// SIMATIC S7-200 SMART project (STEP 7-Micro/WIN SMART), CPU ST40

SYMBOL_TABLE Table 1
Counter_1        C1
CON_Done         M0.0
CON_Busy         M0.1
CON_Error        M0.2
CON_Stat         MB1
SEND_Done        M2.0
SEND_Busy        M2.1
SEND_Error       M2.2
SEND_Stat        MB3
END_SYMBOL_TABLE

SYMBOL_TABLE System Symbols
Always_On        SM0.0    // Always ON
First_Scan_On    SM0.1    // ON for the first scan cycle only
Clock_1s         SM0.5    // Clock pulse that is ON for 0.5 s, OFF for 0.5 s, for a duty cycle time of 1 s.
END_SYMBOL_TABLE

ORGANIZATION_BLOCK MAIN:OB1
TITLE=Program Comments
BEGIN
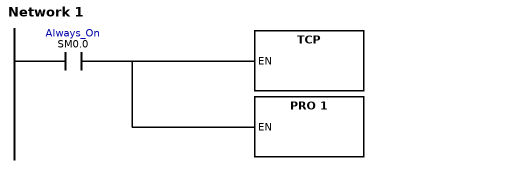
Network 1
LD     Always_On:SM0.0
CALL   TCP:SBR12
CALL   PRO 1:SBR0
END_ORGANIZATION_BLOCK

SUBROUTINE_BLOCK PRO 1:SBR0
TITLE=Subroutine Comments
BEGIN
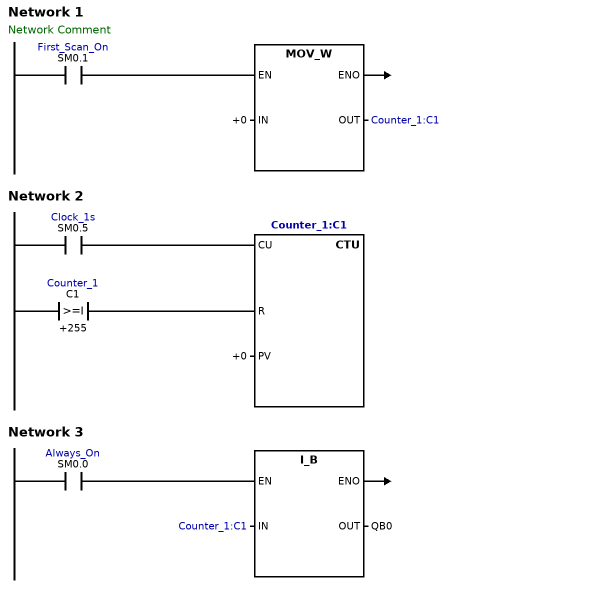
Network 1
// Network Comment
LD     First_Scan_On:SM0.1
MOVW   +0, Counter_1:C1
Network 2
LD     Clock_1s:SM0.5
LDW>=  Counter_1:C1, +255
CTU    Counter_1:C1, +0
Network 3
LD     Always_On:SM0.0
ITB    Counter_1:C1, QB0
END_SUBROUTINE_BLOCK

// SBR10: protected block, not included

// SBR11: protected block, not included

SUBROUTINE_BLOCK TCP:SBR12
TITLE=Subroutine Comments
BEGIN
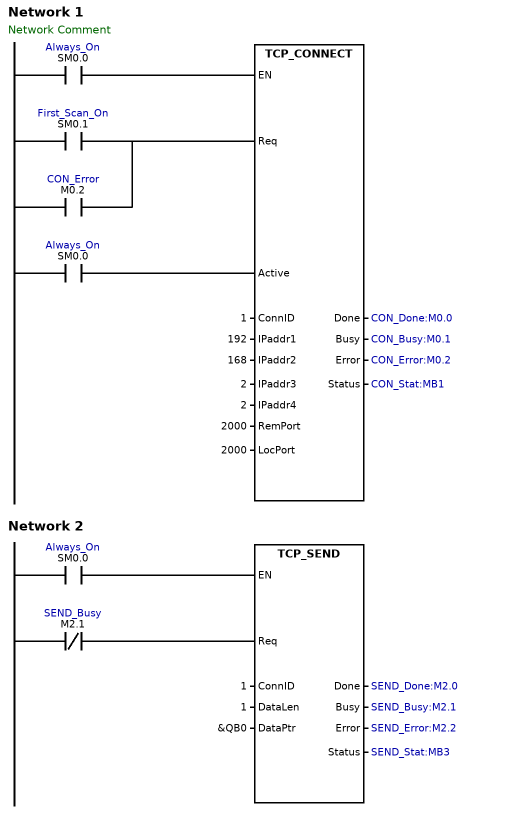
Network 1
// Network Comment
LD     Always_On:SM0.0
=      L60.0
LD     First_Scan_On:SM0.1
O      CON_Error:M0.2
=      L63.7
LD     Always_On:SM0.0
=      L63.6
LD     L60.0
CALL   TCP_CONNECT:SBR10, L63.7, L63.6, 1, 192, 168, 2, 2, 2000, 2000, CON_Done:M0.0, CON_Busy:M0.1, CON_Error:M0.2, CON_Stat:MB1
Network 2
LD     Always_On:SM0.0
=      L60.0
LDN    SEND_Busy:M2.1
=      L63.7
LD     L60.0
CALL   TCP_SEND:SBR11, L63.7, 1, 1, &QB0, SEND_Done:M2.0, SEND_Busy:M2.1, SEND_Error:M2.2, SEND_Stat:MB3
END_SUBROUTINE_BLOCK
